TYPE CmpConvStopConfig :
STRUCT
	
	HandshakeUpstream: BOOL;
	HasLocate: BOOL; 
	DoesWorkRequest: BOOL;
	HandshakeDownstream: BOOL;
	BufferOnlyOneInMotion: BOOL;
	BufferArrivalFault: BOOL;
	RemoteBufferSensor: BOOL;
	DepartStopFaultTime: TIME;
	TimeSpacingMinimum: TIME;
	BufferArrivalFaultTime: TIME;
	PuckSensorOnTime: TIME;
	PuckSensorOffTime: TIME;
	LocateOpenedSensorOnTime: TIME;
	LocateClosedSensorOnTime: TIME;
	BufferSensorOnTime: TIME;
	BufferSensorOffTime: TIME;

END_STRUCT
END_TYPE

(* stored: Version 1.1.0.1, ProductVersion 3.1.4024.6
   DUT CmpConvStopConfig: Id {5efdd4c0-4e71-4e17-aca6-895063a7ae2e} *)
